{attribute 'no_check'}
FUNCTION_BLOCK AxDriveBase EXTENDS EcSlaveInfoDataExt IMPLEMENTS I_AxDriveBase
VAR CONSTANT         	
END_VAR  
VAR_INPUT
	rAxis													:	REFERENCE TO AXIS_REF := 0; //Reference to NC-Axis REF
END_VAR                     					
VAR_IN_OUT                  					
END_VAR                     					
VAR_OUTPUT                  					
	Fault													:	BOOL; (* Drive Error *)
	SwitchedOn												:	BOOL; (* Drive enabled *)
	Ready													:	BOOL; (* Drive Ready *)
{attribute 'displaymode':='binary'}    
	Statusword										AT %I* 	:	UINT; //Link to the drive status word after linking the NC
	Channel											AT %I*	:	USINT;
END_VAR                     					                   					
VAR                         				

END_VAR
VAR

(* Cache *********************************************************************)
	State													:	INT; //State machine 

(* Timer ********************************************************************************)

(* Trigger ******************************************************************************)

(* Instance ****************************************************************************)
	
(* Dummy Speicher **********************************************************)
END_VAR

	(* Drive base information															*)
	(************************************************************************************)
	
	SUPER^();

PROPERTY PUBLIC rAxDrive : REFERENCE TO AxDriveBase
GET
rAxDrive REF= This^;
END_GET
END_PROPERTY

PROPERTY Public rInfoData : reference to EcSlaveInfoData
GET
rInfoData REF= THis^;
END_GET
END_PROPERTY

END_FUNCTION_BLOCK

(* stored: Version 1.1.0.1, ProductVersion 3.1.4024.12
   POU AxDriveBase: Id {3d5d5ecc-04ba-4602-80b9-5abf2c607d74}, SpecialFunc None
   Property rAxDrive: Id {1fe46542-f8ae-4e3c-949f-8e4d0fd7a242}
   Get Get: Id {6592a583-77a1-4112-b887-94a74f6e784a}
   Property rInfoData: Id {d5d38b8b-816d-4578-a893-bedfc8cf1f99}
   Get Get: Id {7f7cebab-97b3-48cc-9ceb-80472c5a9d00} *)
